// TIA Portal V20 export
TYPE "typeCmControlNode"
// stored: Namespace Unit1.Em13
   STRUCT
      interlock : "Unit1.Em13.typeCmControlNodeInterlock";
      command : "Unit1.Em13.typeCmControlNodeCommand";
      softcam : "Unit1.Em13.typeCmControlNodeSoftCam";
      brakeTest : "Unit1.Em13.typeCmControlNodeBrakeTest";
   END_STRUCT;
END_TYPE
